FUNCTION CheckDivByte : BYTE
VAR_INPUT
    divisor : BYTE;
END_VAR
VAR
END_VAR

IF divisor = 0 THEN
    CheckDivByte := 1;(**)
ELSE
    CheckDivByte := divisor;
END_IF

END_FUNCTION

(* stored: Version 1.1.0.1, ProductVersion 3.1.4024.12
   POU CheckDivByte: Id {058d4a0a-2b72-401f-9ff1-b480bb2c5c86}, SpecialFunc None *)
